Staubli VAL3: showMessage.pgx

program showMessage()
  local string l_sMessage
begin
  // INIT
  bShowMessage=false
  // look for the esStatus
  if esStatus()==2
    call language:message(l_sMessage,222)
    bShowMessage=true
  else
    // look for the Working Mode and power in SimulMode
    if cycleStatus:bSimulation or bMoveToPoint
      if !isPowered() and cycleStatus:nWorkingMode!=4
        call language:message(l_sMessage,201)
        bShowMessage=true
      elseIf cycleStatus:nWorkingStatus!=0
        // PRESS MOVE HOLD
        call language:message(l_sMessage,203)
        if cycleStatus:nWorkingMode==1
          switch cycleStatus:nWorkingStatus
            case 2
              // JOINT
              call language:message(l_sMessage,140)
            break
            case 3
              // WORLD
              call language:message(l_sMessage,141)
            break
            case 4
              // TOOL
              call language:message(l_sMessage,142)
            break
            case 5
              // POINT
              call language:message(l_sMessage,143)
            break
          endSwitch
        endIf
        bShowMessage=true
      elseIf bStepping
        l_sMessage=" STEPPING ..."
        bShowMessage=true
      endIf
    endIf
  endIf
  //
  if bShowMessage
    call use:timerDialog(l_sMessage,0)
  endIf
end
